INTERFACE I_Valve

METHOD MoveToHome : BOOL
VAR_INPUT
END_VAR
END_METHOD

METHOD MoveToWork : BOOL
VAR_INPUT
END_VAR
END_METHOD

END_INTERFACE

(* stored: Version 1.1.0.1
   Itf I_Valve: Id {7536f8e8-3738-4ee5-9e85-b5edf435218a}
   Method MoveToHome: Id {b8f49c62-f4c0-45b2-9631-25c7b153820d}
   Method MoveToWork: Id {4421bf81-2d66-4e10-8469-b76405e3ef81} *)
